FUNCTION_BLOCK ABSTRACT CUBaseAutomat EXTENDS TcoTaskedSequencer
VAR
END_VAR

PROPERTY PRIVATE BaseStation : REFERENCE TO CUBase
GET
VAR
    _station : POINTER TO CUBase;
END_VAR
IF __QUERYPOINTER(Parent, _station) THEN // Check if _Parent is Station001
    BaseStation REF= _station^;              // If the check is successful dereference a pointer. simlar to THIS^ or SUPER^
END_IF
END_GET
END_PROPERTY

END_FUNCTION_BLOCK

(* stored: Version 1.1.0.1
   POU CUBaseAutomat: Id {f34497ee-0ea8-4948-9690-a8151302d35b}, SpecialFunc None
   Property BaseStation: Id {2f34bbe0-ae77-4424-96f8-d75571b12d83}
   Get Get: Id {5ff633c4-e770-483e-b525-87fa0c0de322} *)
